(* IEC 61131-3 sources: RL_MAR/experiments/comparison/llm4plc/results/deepseek-ai-DeepSeek-V3.2_20260506_104945/20260506_114017, 4 files *)

(* ---- generated_code_iteration_0.st ---- *)
START_ST
TYPE POINT :
STRUCT
    X : INT;
    Y : INT;
END_STRUCT
END_TYPE

FUNCTION_BLOCK FB_PointOperations
VAR_INPUT
    INPUT_VAR2 : INT := 7;
END_VAR
VAR_OUTPUT
    OUTPUT_VAR1 : POINT;
    OUTPUT_VAR3 : POINT;
END_VAR
VAR
    VAR2 : INT;
END_VAR

    VAR2 := INPUT_VAR2;
    OUTPUT_VAR1.X := 1;
    OUTPUT_VAR1.Y := 2;
    OUTPUT_VAR3.X := 100;
    OUTPUT_VAR3.Y := -7000;

END_FUNCTION_BLOCK
END_ST

(* ---- generated_code_iteration_1.st ---- *)
START_REASON
The validation feedback indicates that the CODESYS compiler validation failed with the error "未知的类型: 'POINT'" (unknown type: 'POINT'). This error occurs because the user-defined type POINT is defined outside the FUNCTION_BLOCK, but in CODESYS, type definitions must be placed in a specific location, typically in a separate type definition section or within the same compilation unit. In Structured Text for CODESYS, type definitions like POINT should be defined before the FUNCTION_BLOCK, but they must be properly scoped. Since the feedback suggests the code failed CODESYS validation, I need to ensure the type definition is correctly integrated. In CODESYS, type definitions are often placed in a DUT (Data Unit Type) or directly in the same POU (Program Organization Unit) if allowed. However, based on common CODESYS practices, I should define the POINT type as a STRUCT within the same context, but the error suggests it's not recognized. I will move the type definition inside the FUNCTION_BLOCK or ensure it's properly declared. Alternatively, I can define it as a local type within the FUNCTION_BLOCK using TYPE...END_TYPE inside the VAR section, but that might not be standard. Instead, I'll define POINT as a global type by placing it before the FUNCTION_BLOCK and ensure it's correctly referenced. The original code defined POINT with TYPE...END_TYPE, which should be valid, but CODESYS might require it to be in a DUT. To fix this, I'll keep the type definition external but ensure it's properly formatted. I'll also correct the variable declarations to use END_VAR appropriately as per the task description.
END_REASON

START_ST
TYPE POINT :
STRUCT
    X : INT;
    Y : INT;
END_STRUCT
END_TYPE

FUNCTION_BLOCK FB_PointOperations
VAR_INPUT
    INPUT_VAR2 : INT := 7;
END_VAR
VAR_OUTPUT
    OUTPUT_VAR1 : POINT;
    OUTPUT_VAR3 : POINT;
END_VAR
VAR
    VAR2 : INT;
END_VAR

    VAR2 := INPUT_VAR2;
    OUTPUT_VAR1.X := 1;
    OUTPUT_VAR1.Y := 2;
    OUTPUT_VAR3.X := 100;
    OUTPUT_VAR3.Y := -7000;

END_FUNCTION_BLOCK
END_ST

(* ---- generated_code_iteration_2.st ---- *)
START_REASON
The validation feedback indicates an encoding issue with the CODESYS compiler check, specifically a 'gbk' codec error due to an illegal multibyte sequence at position 110. This suggests that the code contains non-ASCII characters or invalid byte sequences that cannot be decoded properly. In the previous ST code, all characters appear to be ASCII (e.g., letters, numbers, symbols), but there might be hidden or special characters introduced during copy-pasting or formatting. To resolve this, I need to ensure the code uses only standard ASCII characters and avoid any non-printable or extended characters. I will rewrite the code from scratch, ensuring it is clean and free of encoding issues. Additionally, I will maintain the FUNCTION_BLOCK structure, use END_VAR correctly, and define the POINT type appropriately. Since the feedback does not specify other errors, I will assume the structural aspects are correct but need encoding fixes. I will generate the code with plain ASCII text.
END_REASON

START_ST
TYPE POINT :
STRUCT
    X : INT;
    Y : INT;
END_STRUCT
END_TYPE

FUNCTION_BLOCK FB_PointOperations
VAR_INPUT
    INPUT_VAR2 : INT := 7;
END_VAR
VAR_OUTPUT
    OUTPUT_VAR1 : POINT;
    OUTPUT_VAR3 : POINT;
END_VAR
VAR
    VAR2 : INT;
END_VAR

    VAR2 := INPUT_VAR2;
    OUTPUT_VAR1.X := 1;
    OUTPUT_VAR1.Y := 2;
    OUTPUT_VAR3.X := 100;
    OUTPUT_VAR3.Y := -7000;

END_FUNCTION_BLOCK
END_ST

(* ---- generated_code_iteration_3.st ---- *)
START_REASON
The validation feedback indicates that the CODESYS compiler does not recognize the type 'POINT'. This is likely because the TYPE definition for POINT is placed outside the FUNCTION_BLOCK, but in CODESYS, type definitions might need to be declared within the appropriate scope or in a separate DUT (Data Unit Type) section. In structured text for CODESYS, user-defined types like POINT are typically defined in a separate type declaration area (e.g., in a DUT), not directly within the FUNCTION_BLOCK code. However, since the task requires generating a complete ST code block, I should define the POINT type inside the FUNCTION_BLOCK or ensure it is properly scoped. Based on common CODESYS practices, I can define the POINT structure as a local type within the FUNCTION_BLOCK using TYPE...END_TYPE inside the VAR section or as a global definition, but for simplicity and to avoid scope issues, I will move the POINT definition to a DUT-like section at the top of the code, before the FUNCTION_BLOCK. This should make it accessible. I will restructure the code to include the type definition in a way that CODESYS accepts, typically by placing it in a TYPE block before the FUNCTION_BLOCK. I will also ensure all variable declarations use END_VAR correctly and maintain ASCII-only characters to prevent encoding errors.
END_REASON

START_ST
TYPE POINT :
STRUCT
    X : INT;
    Y : INT;
END_STRUCT
END_TYPE

FUNCTION_BLOCK FB_PointOperations
VAR_INPUT
    INPUT_VAR2 : INT := 7;
END_VAR
VAR_OUTPUT
    OUTPUT_VAR1 : POINT;
    OUTPUT_VAR3 : POINT;
END_VAR
VAR
    VAR2 : INT;
END_VAR

    VAR2 := INPUT_VAR2;
    OUTPUT_VAR1.X := 1;
    OUTPUT_VAR1.Y := 2;
    OUTPUT_VAR3.X := 100;
    OUTPUT_VAR3.Y := -7000;

END_FUNCTION_BLOCK
END_ST
